FUNCTION_BLOCK FB_PC_OneLink_GasSensor EXTENDS FB_PC_OneLink_Base
VAR_INPUT
END_VAR
VAR_OUTPUT
END_VAR
VAR
END_VAR


// XMEAS RANGES
G_PARAMS.A_FLOW_MAX 	:=20.0;
G_PARAMS.D_FLOW_MAX		:=20.0;

G_PARAMS.A_FLOW_MIN 	:=0.0;
G_PARAMS.D_FLOW_MIN		:=0.0;

// execute the signal conversion
SUPER^();

END_FUNCTION_BLOCK

(* stored: Version 1.1.0.1, ProductVersion 3.1.4020.12
   POU FB_PC_OneLink_GasSensor: Id {5f9f9655-a526-448d-b863-035adc563453}, SpecialFunc None *)
